TYPE (* A Structure with 2 BOOLS *)
  (* Version 1.0, 2024-02-21, Franz Höpfinger, HR Agrartechnik GmbH *)
  ST02B : STRUCT
    B_00 : BOOL; (* BIT 00 *)
    B_01 : BOOL; (* BIT 01 *)
  END_STRUCT;
END_TYPE
